FUNCTION_BLOCK FB_AxisWriteNC
VAR_INPUT
END_VAR
VAR_OUTPUT
END_VAR
VAR
END_VAR

END_FUNCTION_BLOCK

(* stored: Version 1.1.0.1, ProductVersion 3.1.4022.12
   POU FB_AxisWriteNC: Id {f7f47c17-7b1c-42c7-9653-657995f4107e}, SpecialFunc None *)
